// TIA Portal V17 export
FUNCTION "FC_FanGasControl" : Void   // FC, LAD
{ S7_Optimized_Access := 'TRUE' }
BEGIN

REGION Network 1: 风机运行联锁
   // 风机运行按接通且风机故障反馈未动作时，驱动风机运行线圈
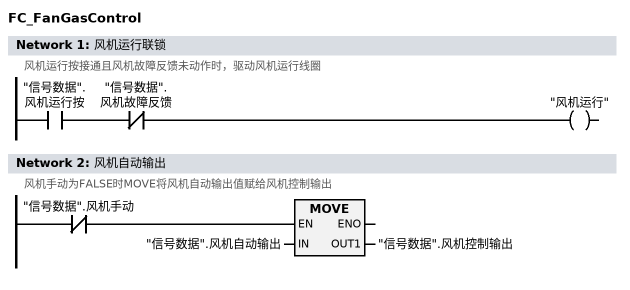
   RUNG wire#powerrail
      Contact( "信号数据".风机运行按 )
      I_Contact( "信号数据".风机故障反馈 )
      Coil( "风机运行" )
   END_RUNG
   // the same network as SCL:
   "风机运行" := "信号数据".风机运行按 AND NOT "信号数据".风机故障反馈;
END_REGION

REGION Network 2: 风机自动输出
   // 风机手动为FALSE时MOVE将风机自动输出值赋给风机控制输出
   RUNG wire#powerrail
      I_Contact( "信号数据".风机手动 )
      { S7_GenerateENO := "TRUE" } Move(in := "信号数据".风机自动输出, out1 => "信号数据".风机控制输出)
   END_RUNG
   // the same network as SCL:
   IF NOT "信号数据".风机手动 THEN "信号数据".风机控制输出 := "信号数据".风机自动输出; END_IF;
END_REGION
END_FUNCTION
